FUNCTION_BLOCK PtDateTime IMPLEMENTS I_PtDateTime
VAR_INPUT
END_VAR
VAR_OUTPUT
END_VAR
VAR
	_Year : DINT;
	_Month : DINT;
	_Day : DINT;
	_Hour : DINT;
	_Minute : DINT;
	_Second : DINT;
	_Microsecond : DINT;
	_TimeZone : DINT;
	
END_VAR

PROPERTY Day : DINT
GET
Day := _Day;
END_GET
SET
_Day := Day;
END_SET
END_PROPERTY

METHOD Diff : I_PtInterval
VAR_INPUT
	TargetDateTime : PtDateTime;
END_VAR
//Diff.Set(THIS^,TargetDateTime,TRUE);
Pendulum._interval.Set(THIS^,TargetDateTime,TRUE);
Diff := Pendulum._interval;
END_METHOD

PROPERTY Hour : DINT
GET
Hour := _Hour;
END_GET
SET
_Hour := Hour;
END_SET
END_PROPERTY

PROPERTY Microsecond : DINT
GET
Microsecond := _Microsecond;
END_GET
SET
_Microsecond := Microsecond;
END_SET
END_PROPERTY

PROPERTY Minute : DINT
GET
Minute := _Minute;
END_GET
SET
_Minute := Minute;
END_SET
END_PROPERTY

PROPERTY Month : DINT
GET
Month := _Month;
END_GET
SET
_Month := Month;
END_SET
END_PROPERTY

PROPERTY Second : DINT
GET
Second := _Second;
END_GET
SET
_Second := Second;
END_SET
END_PROPERTY

METHOD Set //: PtDateTime
VAR_INPUT
	Year : DINT;
	Month : DINT;
	Day : DINT;
	Hour : DINT;
	Minute : DINT;
	Second : DINT;
	Microsecond : DINT;
	TimeZone : DINT;
END_VAR
THIS^._Year := Year;
THIS^._Month := Month;
THIS^._Day := Day;
THIS^._Hour := Hour;
THIS^._Minute := Minute;
THIS^._Second := Second;
THIS^._Microsecond := Microsecond;
THIS^._TimeZone := TimeZone;
END_METHOD

PROPERTY TimeZone : DINT
GET
TimeZone := _TimeZone;
END_GET
SET
_TimeZone := TimeZone;
END_SET
END_PROPERTY

PROPERTY Year : DINT
GET
Year := _Year;
END_GET
SET
_Year := Year;
END_SET
END_PROPERTY

END_FUNCTION_BLOCK

(* stored: Version 1.1.0.1, ProductVersion 3.1.4024.12
   POU PtDateTime: Id {9c733479-bff0-434a-9ceb-c663fdd00bd4}, SpecialFunc None
   Property Day: Id {fe9e7205-9b44-4e81-af58-a74ce464bc7d}
   Get Get: Id {dd281ff5-75a6-4779-b0d7-a446712244b9}
   Set Set: Id {594675a8-789f-4319-9b2b-e9e0cde633ed}
   Method Diff: Id {426f9979-572f-4a55-a26e-46110bd175bd}
   Property Hour: Id {777aaebf-7dac-408f-be17-ce9179131ffb}
   Get Get: Id {ab96bd36-c84e-4bfa-aab2-264fcc48045d}
   Set Set: Id {61650289-5b4c-46a7-90f2-0e37a600c51d}
   Property Microsecond: Id {6acf02b3-65b3-4953-887a-07b4d3bc6200}
   Get Get: Id {d46e4975-d006-4d3b-b68d-fa61a13cccb3}
   Set Set: Id {dfa1a0fc-d2a3-410e-9810-26eeb44395a9}
   Property Minute: Id {87fd9fbe-2977-487f-a486-30a4a9721474}
   Get Get: Id {a45730f7-948c-4d9e-9a93-77ae9185fb41}
   Set Set: Id {37489453-f520-4e2a-b3cc-a97e9c5fd303}
   Property Month: Id {7809000c-0ace-4d5a-bda4-718643e25354}
   Get Get: Id {1d31989b-e957-427d-90e1-6dbcb6c268e3}
   Set Set: Id {9c508cee-52fc-436d-be50-b4508a1391d5}
   Property Second: Id {ee116c1b-0562-4572-930d-4ff27ed39f9a}
   Get Get: Id {b899b81d-c388-43f6-9671-533d46f8dd11}
   Set Set: Id {d6582638-188c-425a-9074-f062a1cd6473}
   Method Set: Id {8cc1b098-ebe9-4963-8754-fc998fa77f3e}
   Property TimeZone: Id {e19480f2-1dce-46fd-b540-5f4d8f72a740}
   Get Get: Id {a62405e9-d3dd-4d3a-a783-2ef8d6d15aa3}
   Set Set: Id {47188b50-955b-4522-b9be-e72d93aa72e2}
   Property Year: Id {f90e6b7f-e4e5-4d6d-9541-0cf108a9e464}
   Get Get: Id {1057d9f6-c06f-40be-9e9e-29e1939bf543}
   Set Set: Id {8ddef1ea-0b29-4f80-8bb5-f55d069a6a02} *)
